FUNCTION_BLOCK FB_Emitter

VAR_INPUT
	LIGHTARRAY : BOOL;
	SALECAJA: BOOL;
	RESET : BOOL;
END_VAR

VAR_OUTPUT
	CINTA : BOOL;
END_VAR

VAR
	bRTrigReset: R_TRIG;
	tRTrigEmitter: R_TRIG;
END_VAR

(* Este FB se encarga de controlar la activaicón y desactivación de los roller
mientras haya o no haya una caja a la espera *)
tRTrigEmitter(CLK:= LIGHTARRAY, Q=> RESET);

RESET := FALSE;

IF NOT SALECAJA THEN
	IF NOT LIGHTARRAY THEN
		CINTA := TRUE;	
	END_IF
	
	IF LIGHTARRAY THEN
		CINTA := FALSE;
	END_IF
END_IF

END_FUNCTION_BLOCK

(* stored: Version 1.1.0.1, ProductVersion 3.1.4024.12
   POU FB_Emitter: Id {0941df9b-1ff2-48dc-8131-9854314bbfe4}, SpecialFunc None *)
